(* PLC project v0.6.02_RefactorGateAndTest.project, CODESYS CODESYS V3.5 SP19 Patch 1 *)
(* stored: creationDateTime 2026-08-14T10:10:49.359610, modificationDateTime 2026-08-14T10:10:49.359610 *)

(* ═══════════════════════════════════════════════════════════════ 🔧 ST_CycleCfg — Configuration du cycle semi-automatique 🐛 T66 : SetDepth_M/SetOffset_M protégés par persistance GVL_PERSISTENT (voir PRG_SUPERVISION_CFC.st §2/§3) ═══════════════════════════════════════════════════════════════ *)
TYPE ST_CycleCfg : STRUCT
  SetDepth_M : REAL := -12.5;  (* 📐 Profondeur de dragage cible (m, négative) *)
  SetOffset_M : REAL := 1.5;  (* 📐 Décalage cible de fermeture de la benne (m) *)
  Initialized : BOOL := FALSE;  (* 🚦 flag restauration boot *)
END_STRUCT;
END_TYPE

(* ═══════════════════════════════════════════════════════════════ 🌉 FB_CfgPersistBridge_CycleCfg — Pont persistance générique pour ST_CycleCfg ─────────────────────────────────────────────────────────────── 🎯 Voir FB_CfgPersistBridge_SyncCfg.st (Lot 3a) pour la logique de référence — identique, seul le type ST_CycleCfg change. ═══════════════════════════════════════════════════════════════ *)
FUNCTION_BLOCK FB_CfgPersistBridge_CycleCfg
  VAR_OUTPUT
    JustRestored : BOOL;
  END_VAR
  VAR_IN_OUT
    Hmi : ST_CycleCfg;  (* 🖥️ ex. GVL_IHM.Cycle.Cfg *)
    Persist : ST_CycleCfg;  (* 💾 ex. GVL_PERSISTENT._CycleCfgPersist *)
  END_VAR

            

JustRestored := FALSE;
IF NOT Hmi.Initialized THEN
    Hmi := Persist;
    Hmi.Initialized := TRUE;
    JustRestored := TRUE;
ELSE
    Persist := Hmi;
END_IF;

          
END_FUNCTION_BLOCK
